FUNCTION_BLOCK FB_ControlElement4 EXTENDS FB_BaseControlElement IMPLEMENTS ITF_ControlElement4
VAR
	
	itfsenStart			: ITF_IOSensor;
	itfsenEnd			: ITF_IOSensor;	
	itfsenPosition1		: ITF_IOSensor;	
	itfsenPosition2		: ITF_IOSensor;	
END_VAR

METHOD FB_init : BOOL
VAR_INPUT
	bInitRetains : BOOL; // if TRUE, the retain variables are initialized (warm start / cold start)
	bInCopyCode : BOOL;  // if TRUE, the instance afterwards gets moved into the copy code (online change)
	itfsenStart			: ITF_IOSensor;
	itfsenEnd			: ITF_IOSensor;	
	itfsenPosition1		: ITF_IOSensor;	
	itfsenPosition2		: ITF_IOSensor;	
END_VAR
THIS^.itfsenStart					:= itfsenStart;
THIS^.AddComponent (itfComponent	:= itfsenStart);
THIS^.SetText (eLocation 			:= E_BaseLocation.pl, wsDescription := "Nazwa komponentu 1 pl");
THIS^.SetText (eLocation 			:= E_BaseLocation.en, wsDescription := "Nazwa komponentu 1 en");
THIS^.SetText (eLocation 			:= E_BaseLocation.de, wsDescription := "Nazwa komponentu 1 de");
THIS^.itfsenStart.SetName (stName	:= THIS^.GetTexts ());

THIS^.itfsenEnd						:= itfsenEnd;
THIS^.AddComponent (itfComponent	:= itfsenEnd);
THIS^.SetText (eLocation 			:= E_BaseLocation.pl, wsDescription := "Nazwa komponentu 2 pl");
THIS^.SetText (eLocation 			:= E_BaseLocation.en, wsDescription := "Nazwa komponentu 2 en");
THIS^.SetText (eLocation 			:= E_BaseLocation.de, wsDescription := "Nazwa komponentu 2 de");
THIS^.itfsenEnd.SetName (stName	:= THIS^.GetTexts ());

THIS^.itfsenPosition1				:= itfsenPosition1;
THIS^.AddComponent (itfComponent	:= itfsenPosition1);
THIS^.SetText (eLocation 			:= E_BaseLocation.pl, wsDescription := "Nazwa komponentu 3 pl");
THIS^.SetText (eLocation 			:= E_BaseLocation.en, wsDescription := "Nazwa komponentu 3 en");
THIS^.SetText (eLocation 			:= E_BaseLocation.de, wsDescription := "Nazwa komponentu 3 de");
THIS^.itfsenPosition1.SetName (stName	:= THIS^.GetTexts ());

THIS^.itfsenPosition2				:= itfsenPosition2;
THIS^.AddComponent (itfComponent	:= itfsenPosition2);
THIS^.SetText (eLocation 			:= E_BaseLocation.pl, wsDescription := "Nazwa komponentu 4 pl");
THIS^.SetText (eLocation 			:= E_BaseLocation.en, wsDescription := "Nazwa komponentu 4 en");
THIS^.SetText (eLocation 			:= E_BaseLocation.de, wsDescription := "Nazwa komponentu 4 de");
THIS^.itfsenPosition2.SetName (stName	:= THIS^.GetTexts ());
END_METHOD

END_FUNCTION_BLOCK

(* stored: Version 1.1.0.1, ProductVersion 3.1.4024.15
   POU FB_ControlElement4: Id {e2e97afe-1370-47b9-a9aa-42c8b5f3ed77}, SpecialFunc None
   Method FB_init: Id {6a3c40bc-fe3b-48c2-be70-4ae322e99ca8} *)
